(* IEC 61131-3 sources: tree-sitter-structured-text/examples, 4 files *)

(* ---- namespace_and_class.st ---- *)
USING Test.FB;

NAMESPACE TestNamespaceAndClass
    TYPE
        ColorWithValues : (
            RED := 1,
            GREEN := 2,
            BLUE := 3,
            YELLOW := 4) := RED;

        Color : (
            RED,
            GREEN,
            BLUE,
            YELLOW
        );

        TestStruct : STRUCT
            structMember1 : REAL;
            structMember2 : DINT;
        END_STRUCT
    END_TYPE

    {testclass pragma}
    CLASS TestClass
        VAR
            staticVar : BOOL;
        END_VAR

        /// Documentation comment to describe the function
        METHOD PUBLIC TestMethod : INT
            // Input variables of method
            VAR_INPUT
                testInput : REAL;
            END_VAR

            TestMethod := testInput * 2;
        END_METHOD

        METHOD TestCase : INT
            VAR_INPUT
                state : INT;
            END_VAR
            VAR_TEMP
                stateCase : ColorWithValues;
            END_VAR

            CASE state OF
                Color#RED:
                    stateCase := state;
                Color#GREEN:
                    stateCase := state;
                3:
                    stateCase := state;
                Color#YELLOW:
                    stateCase := state;
                ELSE
                    stateCase := 1;
            END_CASE

            TestCase := stateCase;
        END_METHOD
    END_CLASS
END_NAMESPACE

(* ---- function.st ---- *)
FUNCTION TestFunction : BOOL
    VAR_INPUT
        test_input : BOOL;
    END_VAR

    VAR_IN_OUT
        test_in_out : BOOL;
    END_VAR

    IF test_input THEN
        TestFunction := TRUE;
    ELSE
        TestFunction := FALSE;
    END_IF;

    TestFunction := test_in_out;

END_FUNCTION

(* ---- function_block.st ---- *)
NAMESPACE Test.FB
    (*=======================================================================
    Function Block Timed Counter :  Incremental count of the timed interval
    =======================================================================*)
    FUNCTION_BLOCK FB_Timed_Counter
        VAR_INPUT
            Execute         : BOOL := FALSE;        // Trigger signal to begin Timed Counting
            Time_Increment  : REAL := 1.25;         // Enter Cycle Time (Seconds) between counts
            Count_Cycles    : INT  := 20;           // Number of Desired Count Cycles
        END_VAR

        VAR_OUTPUT
            Timer_Done_Bit  : BOOL := FALSE;        // One Shot Bit indicating Timer Cycle Done
            Count_Complete  : BOOL := FALSE;        // Output Bit indicating the Count is complete
            Current_Count   : INT  := 0;            // Accumulating Value of Counter
        END_VAR

        VAR_IN_OUT
            inoutVar : INT;
        END_VAR

        VAR
            CycleTimer      : TON;                  // Timer FB from Command Library
            CycleCounter    : CTU;                  // Counter FB from Command Library
            TimerPreset     : TIME;                 // Converted Time_Increment in Seconds to MS
        END_VAR

        // Start of Function Block programming
        TimerPreset := REAL_TO_TIME(in := Time_Increment) * 1000;

        CycleTimer(
            in := Execute AND NOT CycleTimer.Q,
            pt := TimerPreset);

        Timer_Done_Bit := CycleTimer.Q;

        CycleCounter(
            cu := CycleTimer.Q,
            r := NOT Execute,
            pv := Count_Cycles);

        Current_Count := CycleCounter.cv;
        Count_Complete := CycleCounter.q;

    END_FUNCTION_BLOCK
END_NAMESPACE

(* ---- program.st ---- *)
// PLC configuration
CONFIGURATION DefaultCfg
    VAR_GLOBAL
        b_Start_Stop  : BOOL;         // Global variable to represent a boolean.
        b_ON_OFF      : BOOL;         // Global variable to represent a boolean.
        Start_Stop AT %IX0.0:BOOL;    // Digital   input of the PLC (Address 0.0)
        ON_OFF     AT %QX0.0:BOOL;    // Digital output of the PLC (Address 0.0). (Coil)
    END_VAR

    // Schedule the main program to be executed every 20 ms
    TASK Tick(INTERVAL := t#20ms);

    PROGRAM Main WITH Tick : Monitor_Start_Stop;
END_CONFIGURATION

PROGRAM Monitor_Start_Stop          // Actual Program
    VAR_EXTERNAL
        Start_Stop  : BOOL;
        ON_OFF      : BOOL;
    END_VAR
    VAR                             // Temporary variables for logic handling
        ONS_Trig    : BOOL;
        Rising_ONS  : BOOL;
        Start       : BOOL;
    END_VAR

    // Start of Logic
    // Catch the Rising Edge One Shot of the Start_Stop input
    ONS_Trig    := Start_Stop AND NOT Rising_ONS;

    // if else
    IF Start_Stop THEN
        Start := TRUE;
    ELSE
        Start := FALSE;
    END_IF;

    // Main Logic for Run_Contact -- Toggle ON / Toggle OFF ---
    ON_OFF := (ONS_Trig AND NOT ON_OFF) OR (ON_OFF AND NOT ONS_Trig);

    // Rising One Shot logic
    Rising_ONS := Start_Stop;
END_PROGRAM
